// Mitsubishi GX Works2 project: BluestarPlc 17-06-2023f1   PLC: Q03UDV

PROGRAM MAIN
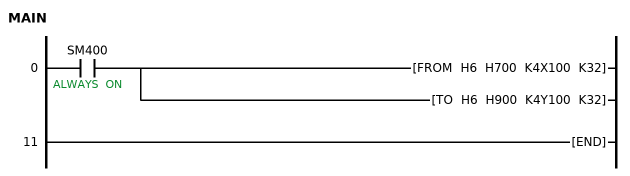
0     LD      SM400  ; ALWAYS  ON
      FROM    H6 H700 K4X100 K32  ; DO1_CMD_ENBLE
      TO      H6 H900 K4Y100 K32  ; DI01_IMSTP
11    END
END_PROGRAM

PROGRAM LOGIC
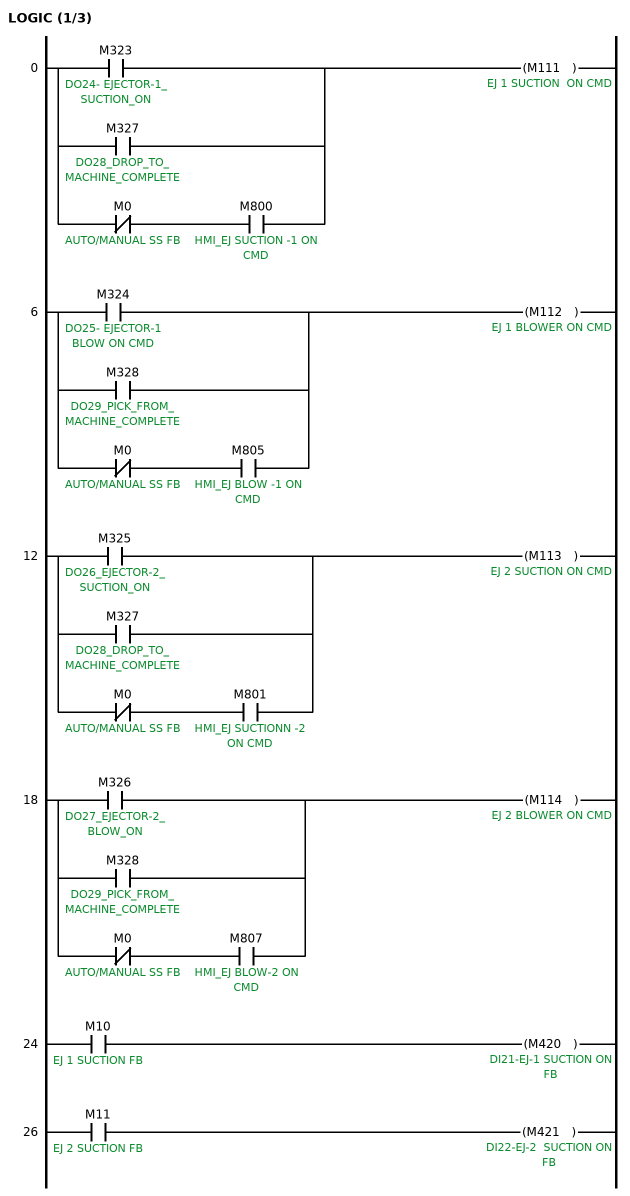
0     LD      M323  ; DO24- EJECTOR-1_SUCTION_ON
      OR      M327  ; DO28_DROP_TO_MACHINE_COMPLETE
      LDI     M0  ; AUTO/MANUAL SS FB
      AND     M800  ; HMI_EJ SUCTION -1 ON CMD
      ORB
      OUT     M111  ; EJ 1 SUCTION  ON CMD
6     LD      M324  ; DO25- EJECTOR-1  BLOW ON CMD
      OR      M328  ; DO29_PICK_FROM_MACHINE_COMPLETE
      LDI     M0  ; AUTO/MANUAL SS FB
      AND     M805  ; HMI_EJ BLOW -1 ON CMD
      ORB
      OUT     M112  ; EJ 1 BLOWER ON CMD
12    LD      M325  ; DO26_EJECTOR-2_SUCTION_ON
      OR      M327  ; DO28_DROP_TO_MACHINE_COMPLETE
      LDI     M0  ; AUTO/MANUAL SS FB
      AND     M801  ; HMI_EJ SUCTIONN -2 ON CMD
      ORB
      OUT     M113  ; EJ 2 SUCTION ON CMD
18    LD      M326  ; DO27_EJECTOR-2_BLOW_ON
      OR      M328  ; DO29_PICK_FROM_MACHINE_COMPLETE
      LDI     M0  ; AUTO/MANUAL SS FB
      AND     M807  ; HMI_EJ BLOW-2 ON CMD
      ORB
      OUT     M114  ; EJ 2 BLOWER ON CMD
24    LD      M10  ; EJ 1 SUCTION FB
      OUT     M420  ; DI21-EJ-1 SUCTION ON FB
26    LD      M11  ; EJ 2 SUCTION FB
      OUT     M421  ; DI22-EJ-2  SUCTION ON FB
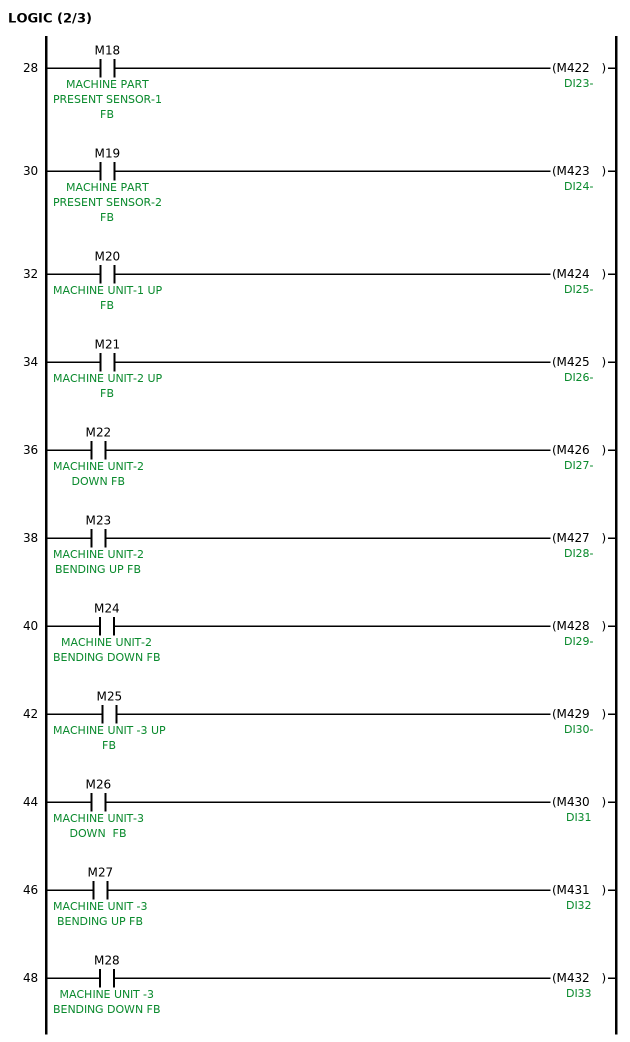
28    LD      M18  ; MACHINE PART PRESENT SENSOR-1 FB
      OUT     M422  ; DI23-
30    LD      M19  ; MACHINE PART PRESENT SENSOR-2 FB
      OUT     M423  ; DI24-
32    LD      M20  ; MACHINE UNIT-1 UP FB
      OUT     M424  ; DI25-
34    LD      M21  ; MACHINE UNIT-2 UP FB
      OUT     M425  ; DI26-
36    LD      M22  ; MACHINE UNIT-2 DOWN FB
      OUT     M426  ; DI27-
38    LD      M23  ; MACHINE UNIT-2 BENDING UP FB
      OUT     M427  ; DI28-
40    LD      M24  ; MACHINE UNIT-2 BENDING DOWN FB
      OUT     M428  ; DI29-
42    LD      M25  ; MACHINE UNIT -3 UP FB
      OUT     M429  ; DI30-
44    LD      M26  ; MACHINE UNIT-3 DOWN  FB
      OUT     M430  ; DI31
46    LD      M27  ; MACHINE UNIT -3 BENDING UP FB
      OUT     M431  ; DI32
48    LD      M28  ; MACHINE UNIT -3 BENDING DOWN FB
      OUT     M432  ; DI33
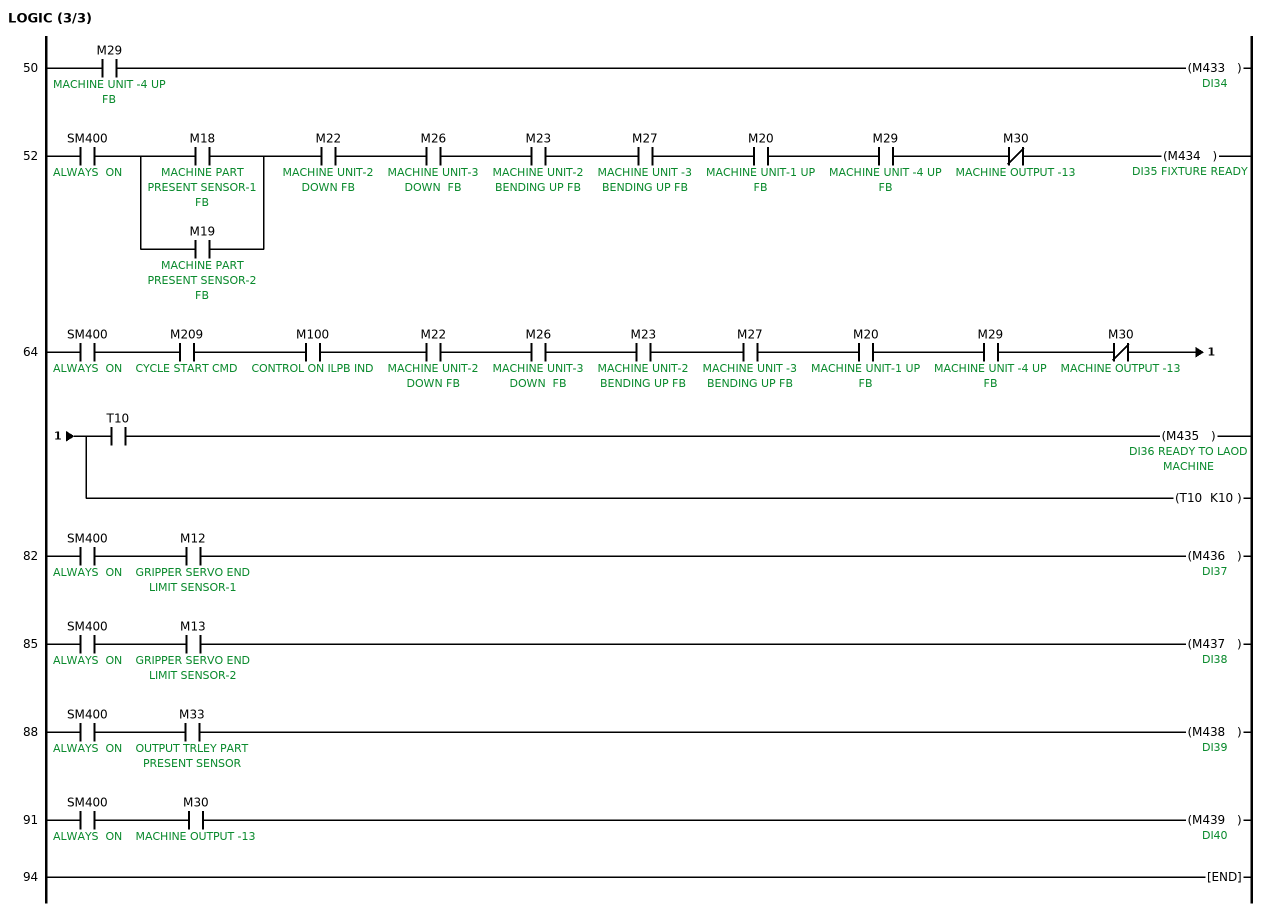
50    LD      M29  ; MACHINE UNIT -4 UP FB
      OUT     M433  ; DI34
52    LD      SM400  ; ALWAYS  ON
      LD      M18  ; MACHINE PART PRESENT SENSOR-1 FB
      OR      M19  ; MACHINE PART PRESENT SENSOR-2 FB
      ANB
      AND     M22  ; MACHINE UNIT-2 DOWN FB
      AND     M26  ; MACHINE UNIT-3 DOWN  FB
      AND     M23  ; MACHINE UNIT-2 BENDING UP FB
      AND     M27  ; MACHINE UNIT -3 BENDING UP FB
      AND     M20  ; MACHINE UNIT-1 UP FB
      AND     M29  ; MACHINE UNIT -4 UP FB
      ANI     M30  ; MACHINE OUTPUT -13
      OUT     M434  ; DI35 FIXTURE READY
64    LD      SM400  ; ALWAYS  ON
      AND     M209  ; CYCLE START CMD
      AND     M100  ; CONTROL ON ILPB IND
      AND     M22  ; MACHINE UNIT-2 DOWN FB
      AND     M26  ; MACHINE UNIT-3 DOWN  FB
      AND     M23  ; MACHINE UNIT-2 BENDING UP FB
      AND     M27  ; MACHINE UNIT -3 BENDING UP FB
      AND     M20  ; MACHINE UNIT-1 UP FB
      AND     M29  ; MACHINE UNIT -4 UP FB
      ANI     M30  ; MACHINE OUTPUT -13
      MPS
      AND     T10
      OUT     M435  ; DI36 READY TO LAOD MACHINE
      MPP
      OUT     T10 K10
82    LD      SM400  ; ALWAYS  ON
      AND     M12  ; GRIPPER SERVO END LIMIT SENSOR-1
      OUT     M436  ; DI37
85    LD      SM400  ; ALWAYS  ON
      AND     M13  ; GRIPPER SERVO END LIMIT SENSOR-2
      OUT     M437  ; DI38
88    LD      SM400  ; ALWAYS  ON
      AND     M33  ; OUTPUT TRLEY PART PRESENT SENSOR
      OUT     M438  ; DI39
91    LD      SM400  ; ALWAYS  ON
      AND     M30  ; MACHINE OUTPUT -13
      OUT     M439  ; DI40
94    END
END_PROGRAM

PROGRAM D-NET
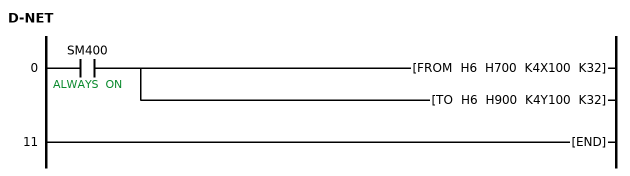
0     LD      SM400  ; ALWAYS  ON
      FROM    H6 H700 K4X100 K32  ; DO1_CMD_ENBLE
      TO      H6 H900 K4Y100 K32  ; DI01_IMSTP
11    END
END_PROGRAM

PROGRAM RBT-IN
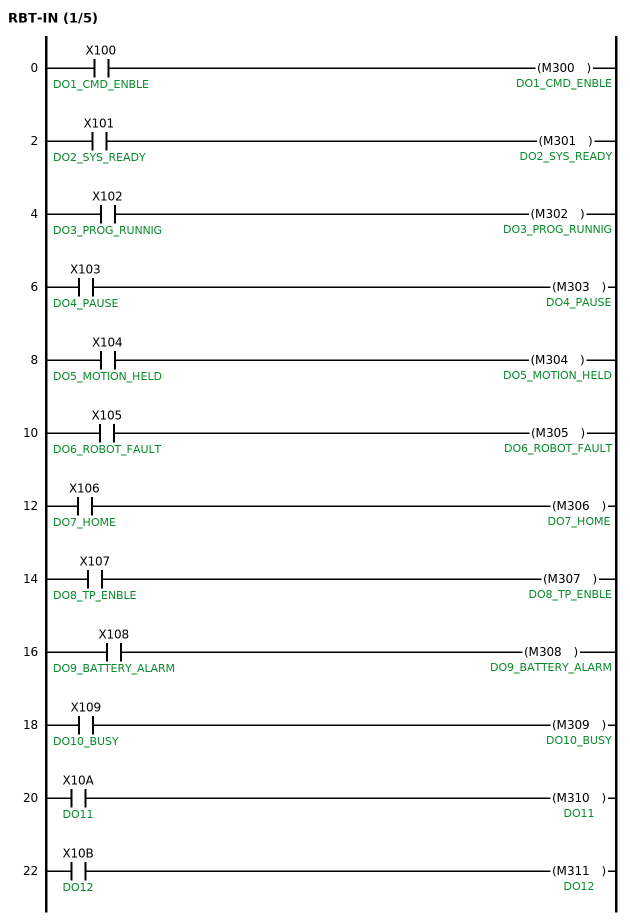
0     LD      X100  ; DO1_CMD_ENBLE
      OUT     M300  ; DO1_CMD_ENBLE
2     LD      X101  ; DO2_SYS_READY
      OUT     M301  ; DO2_SYS_READY
4     LD      X102  ; DO3_PROG_RUNNIG
      OUT     M302  ; DO3_PROG_RUNNIG
6     LD      X103  ; DO4_PAUSE
      OUT     M303  ; DO4_PAUSE
8     LD      X104  ; DO5_MOTION_HELD
      OUT     M304  ; DO5_MOTION_HELD
10    LD      X105  ; DO6_ROBOT_FAULT
      OUT     M305  ; DO6_ROBOT_FAULT
12    LD      X106  ; DO7_HOME
      OUT     M306  ; DO7_HOME
14    LD      X107  ; DO8_TP_ENBLE
      OUT     M307  ; DO8_TP_ENBLE
16    LD      X108  ; DO9_BATTERY_ALARM
      OUT     M308  ; DO9_BATTERY_ALARM
18    LD      X109  ; DO10_BUSY
      OUT     M309  ; DO10_BUSY
20    LD      X10A  ; DO11
      OUT     M310  ; DO11
22    LD      X10B  ; DO12
      OUT     M311  ; DO12
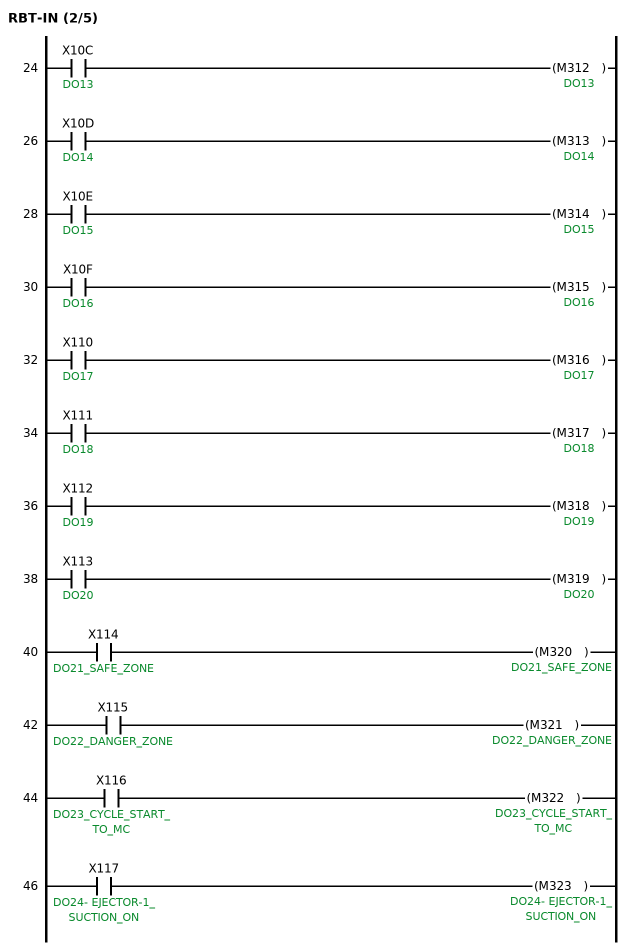
24    LD      X10C  ; DO13
      OUT     M312  ; DO13
26    LD      X10D  ; DO14
      OUT     M313  ; DO14
28    LD      X10E  ; DO15
      OUT     M314  ; DO15
30    LD      X10F  ; DO16
      OUT     M315  ; DO16
32    LD      X110  ; DO17
      OUT     M316  ; DO17
34    LD      X111  ; DO18
      OUT     M317  ; DO18
36    LD      X112  ; DO19
      OUT     M318  ; DO19
38    LD      X113  ; DO20
      OUT     M319  ; DO20
40    LD      X114  ; DO21_SAFE_ZONE
      OUT     M320  ; DO21_SAFE_ZONE
42    LD      X115  ; DO22_DANGER_ZONE
      OUT     M321  ; DO22_DANGER_ZONE
44    LD      X116  ; DO23_CYCLE_START_TO_MC
      OUT     M322  ; DO23_CYCLE_START_TO_MC
46    LD      X117  ; DO24- EJECTOR-1_SUCTION_ON
      OUT     M323  ; DO24- EJECTOR-1_SUCTION_ON
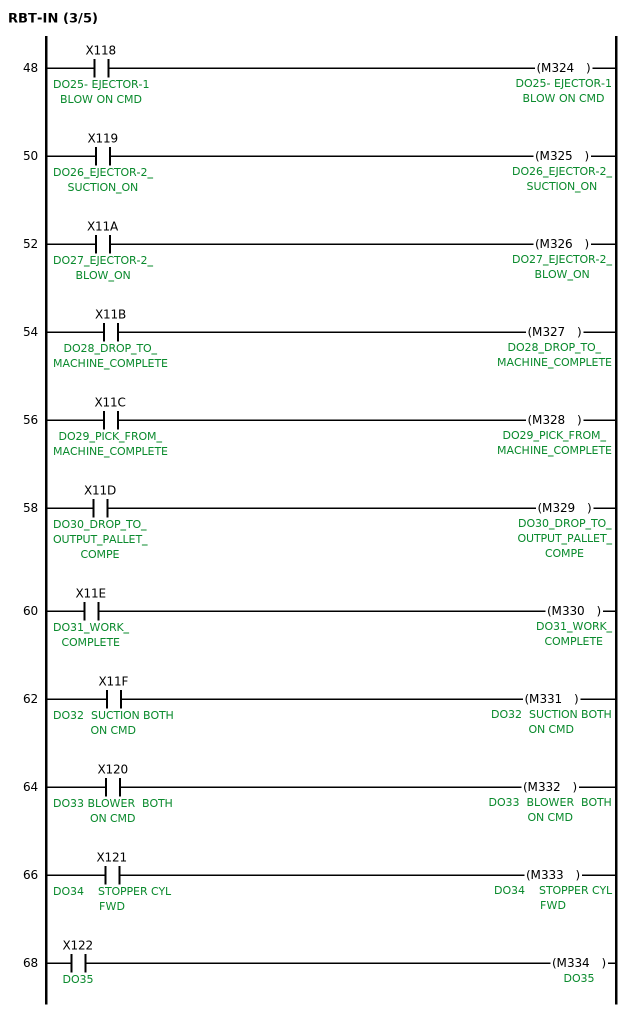
48    LD      X118  ; DO25- EJECTOR-1  BLOW ON CMD
      OUT     M324  ; DO25- EJECTOR-1  BLOW ON CMD
50    LD      X119  ; DO26_EJECTOR-2_SUCTION_ON
      OUT     M325  ; DO26_EJECTOR-2_SUCTION_ON
52    LD      X11A  ; DO27_EJECTOR-2_BLOW_ON
      OUT     M326  ; DO27_EJECTOR-2_BLOW_ON
54    LD      X11B  ; DO28_DROP_TO_MACHINE_COMPLETE
      OUT     M327  ; DO28_DROP_TO_MACHINE_COMPLETE
56    LD      X11C  ; DO29_PICK_FROM_MACHINE_COMPLETE
      OUT     M328  ; DO29_PICK_FROM_MACHINE_COMPLETE
58    LD      X11D  ; DO30_DROP_TO_OUTPUT_PALLET_COMPE
      OUT     M329  ; DO30_DROP_TO_OUTPUT_PALLET_COMPE
60    LD      X11E  ; DO31_WORK_COMPLETE
      OUT     M330  ; DO31_WORK_COMPLETE
62    LD      X11F  ; DO32  SUCTION BOTH ON CMD
      OUT     M331  ; DO32  SUCTION BOTH ON CMD
64    LD      X120  ; DO33 BLOWER  BOTH ON CMD
      OUT     M332  ; DO33  BLOWER  BOTH ON CMD
66    LD      X121  ; DO34    STOPPER CYL FWD
      OUT     M333  ; DO34    STOPPER CYL FWD
68    LD      X122  ; DO35
      OUT     M334  ; DO35
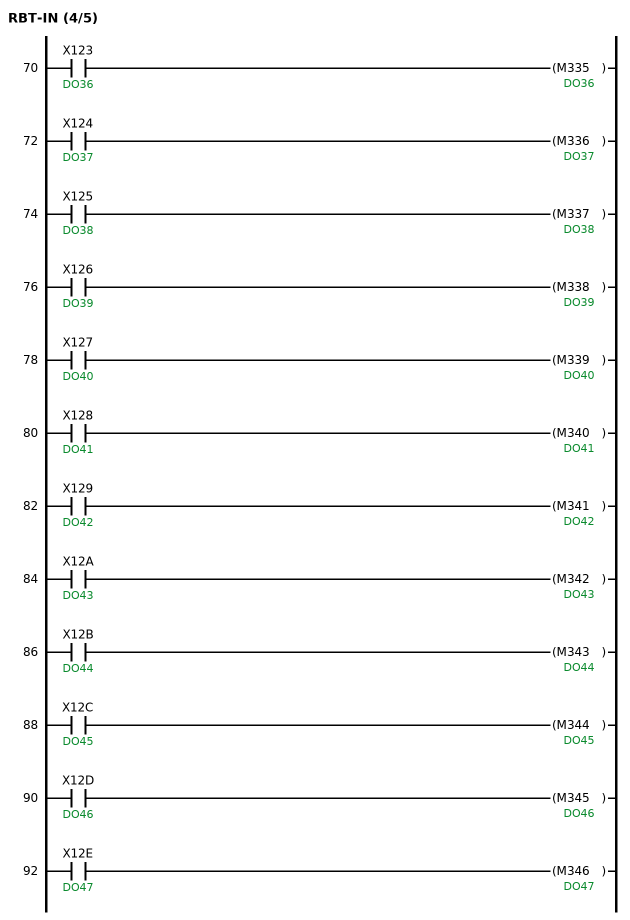
70    LD      X123  ; DO36
      OUT     M335  ; DO36
72    LD      X124  ; DO37
      OUT     M336  ; DO37
74    LD      X125  ; DO38
      OUT     M337  ; DO38
76    LD      X126  ; DO39
      OUT     M338  ; DO39
78    LD      X127  ; DO40
      OUT     M339  ; DO40
80    LD      X128  ; DO41
      OUT     M340  ; DO41
82    LD      X129  ; DO42
      OUT     M341  ; DO42
84    LD      X12A  ; DO43
      OUT     M342  ; DO43
86    LD      X12B  ; DO44
      OUT     M343  ; DO44
88    LD      X12C  ; DO45
      OUT     M344  ; DO45
90    LD      X12D  ; DO46
      OUT     M345  ; DO46
92    LD      X12E  ; DO47
      OUT     M346  ; DO47
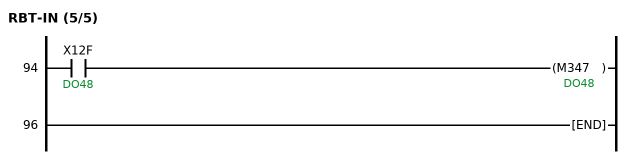
94    LD      X12F  ; DO48
      OUT     M347  ; DO48
96    END
END_PROGRAM

PROGRAM RBT-OUT
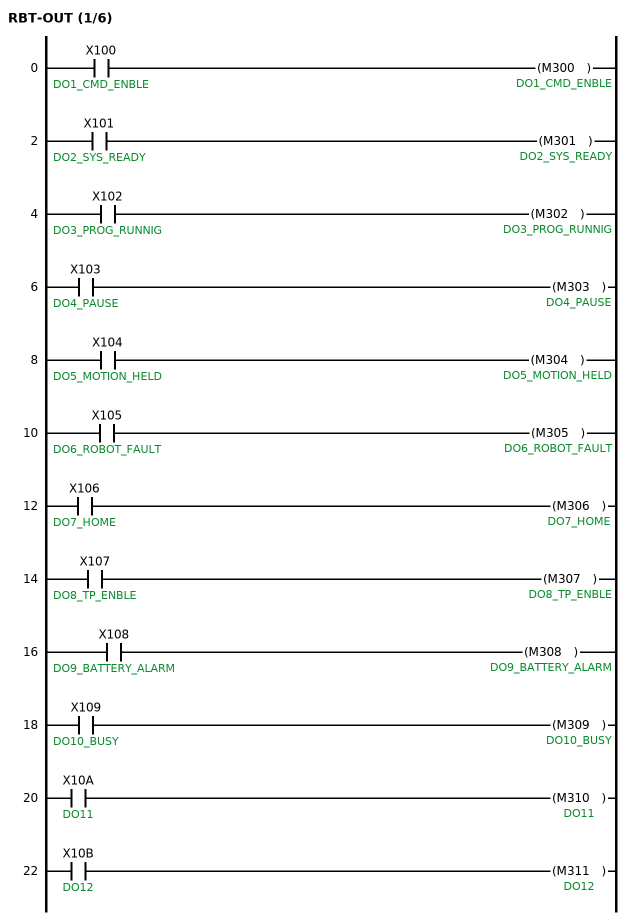
0     LD      X100  ; DO1_CMD_ENBLE
      OUT     M300  ; DO1_CMD_ENBLE
2     LD      X101  ; DO2_SYS_READY
      OUT     M301  ; DO2_SYS_READY
4     LD      X102  ; DO3_PROG_RUNNIG
      OUT     M302  ; DO3_PROG_RUNNIG
6     LD      X103  ; DO4_PAUSE
      OUT     M303  ; DO4_PAUSE
8     LD      X104  ; DO5_MOTION_HELD
      OUT     M304  ; DO5_MOTION_HELD
10    LD      X105  ; DO6_ROBOT_FAULT
      OUT     M305  ; DO6_ROBOT_FAULT
12    LD      X106  ; DO7_HOME
      OUT     M306  ; DO7_HOME
14    LD      X107  ; DO8_TP_ENBLE
      OUT     M307  ; DO8_TP_ENBLE
16    LD      X108  ; DO9_BATTERY_ALARM
      OUT     M308  ; DO9_BATTERY_ALARM
18    LD      X109  ; DO10_BUSY
      OUT     M309  ; DO10_BUSY
20    LD      X10A  ; DO11
      OUT     M310  ; DO11
22    LD      X10B  ; DO12
      OUT     M311  ; DO12
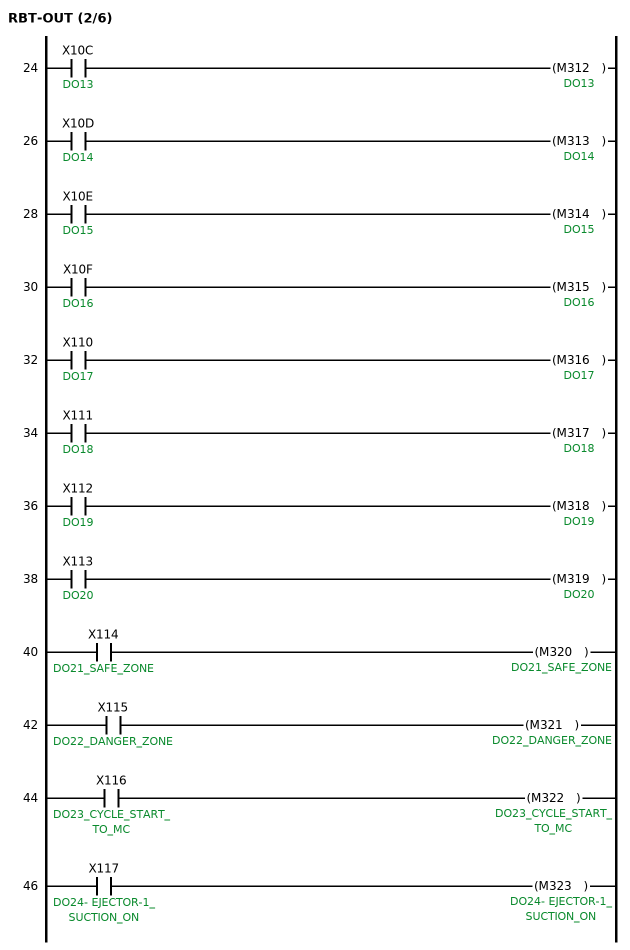
24    LD      X10C  ; DO13
      OUT     M312  ; DO13
26    LD      X10D  ; DO14
      OUT     M313  ; DO14
28    LD      X10E  ; DO15
      OUT     M314  ; DO15
30    LD      X10F  ; DO16
      OUT     M315  ; DO16
32    LD      X110  ; DO17
      OUT     M316  ; DO17
34    LD      X111  ; DO18
      OUT     M317  ; DO18
36    LD      X112  ; DO19
      OUT     M318  ; DO19
38    LD      X113  ; DO20
      OUT     M319  ; DO20
40    LD      X114  ; DO21_SAFE_ZONE
      OUT     M320  ; DO21_SAFE_ZONE
42    LD      X115  ; DO22_DANGER_ZONE
      OUT     M321  ; DO22_DANGER_ZONE
44    LD      X116  ; DO23_CYCLE_START_TO_MC
      OUT     M322  ; DO23_CYCLE_START_TO_MC
46    LD      X117  ; DO24- EJECTOR-1_SUCTION_ON
      OUT     M323  ; DO24- EJECTOR-1_SUCTION_ON
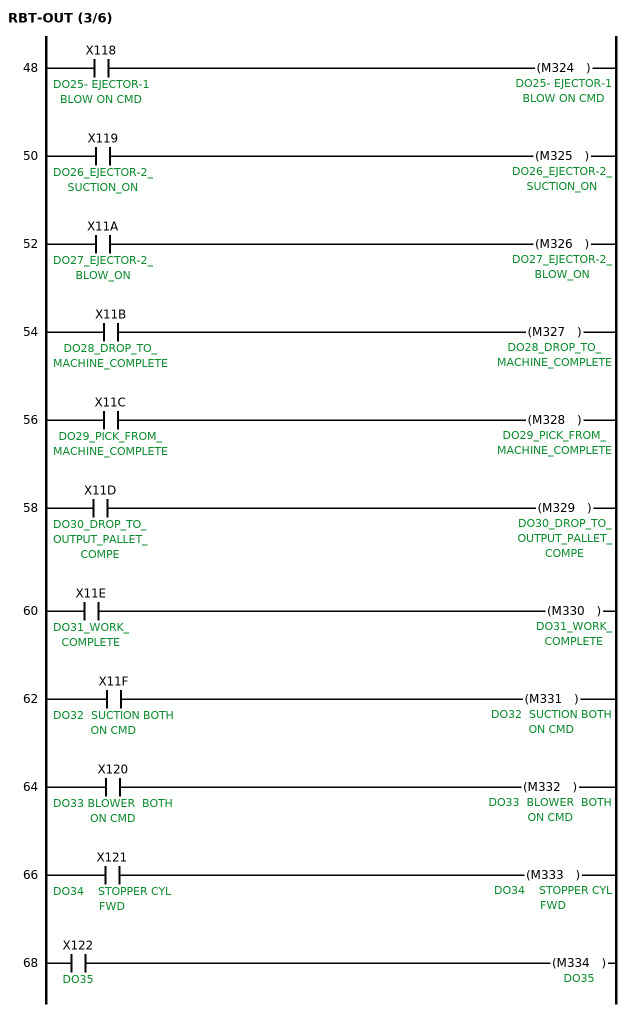
48    LD      X118  ; DO25- EJECTOR-1  BLOW ON CMD
      OUT     M324  ; DO25- EJECTOR-1  BLOW ON CMD
50    LD      X119  ; DO26_EJECTOR-2_SUCTION_ON
      OUT     M325  ; DO26_EJECTOR-2_SUCTION_ON
52    LD      X11A  ; DO27_EJECTOR-2_BLOW_ON
      OUT     M326  ; DO27_EJECTOR-2_BLOW_ON
54    LD      X11B  ; DO28_DROP_TO_MACHINE_COMPLETE
      OUT     M327  ; DO28_DROP_TO_MACHINE_COMPLETE
56    LD      X11C  ; DO29_PICK_FROM_MACHINE_COMPLETE
      OUT     M328  ; DO29_PICK_FROM_MACHINE_COMPLETE
58    LD      X11D  ; DO30_DROP_TO_OUTPUT_PALLET_COMPE
      OUT     M329  ; DO30_DROP_TO_OUTPUT_PALLET_COMPE
60    LD      X11E  ; DO31_WORK_COMPLETE
      OUT     M330  ; DO31_WORK_COMPLETE
62    LD      X11F  ; DO32  SUCTION BOTH ON CMD
      OUT     M331  ; DO32  SUCTION BOTH ON CMD
64    LD      X120  ; DO33 BLOWER  BOTH ON CMD
      OUT     M332  ; DO33  BLOWER  BOTH ON CMD
66    LD      X121  ; DO34    STOPPER CYL FWD
      OUT     M333  ; DO34    STOPPER CYL FWD
68    LD      X122  ; DO35
      OUT     M334  ; DO35
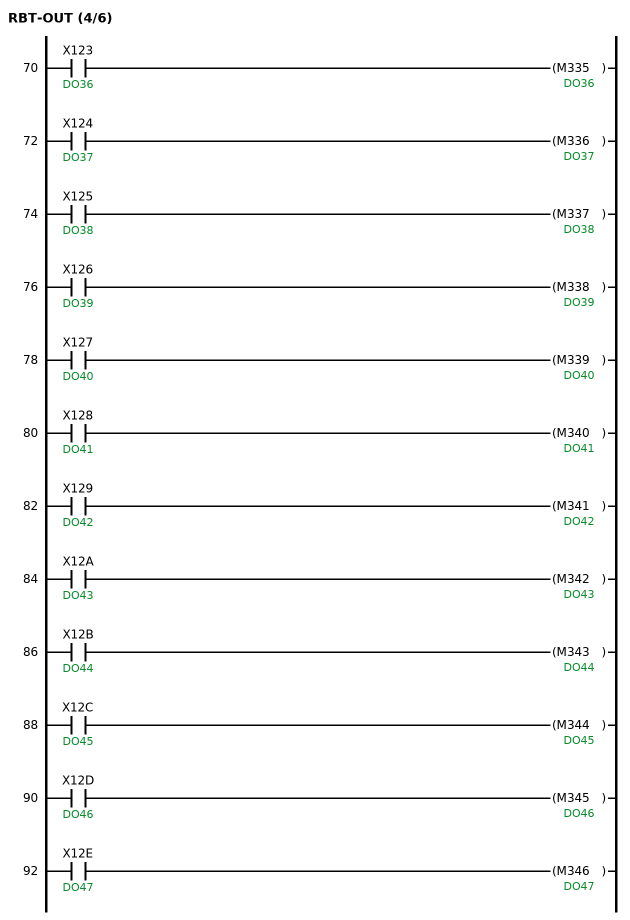
70    LD      X123  ; DO36
      OUT     M335  ; DO36
72    LD      X124  ; DO37
      OUT     M336  ; DO37
74    LD      X125  ; DO38
      OUT     M337  ; DO38
76    LD      X126  ; DO39
      OUT     M338  ; DO39
78    LD      X127  ; DO40
      OUT     M339  ; DO40
80    LD      X128  ; DO41
      OUT     M340  ; DO41
82    LD      X129  ; DO42
      OUT     M341  ; DO42
84    LD      X12A  ; DO43
      OUT     M342  ; DO43
86    LD      X12B  ; DO44
      OUT     M343  ; DO44
88    LD      X12C  ; DO45
      OUT     M344  ; DO45
90    LD      X12D  ; DO46
      OUT     M345  ; DO46
92    LD      X12E  ; DO47
      OUT     M346  ; DO47
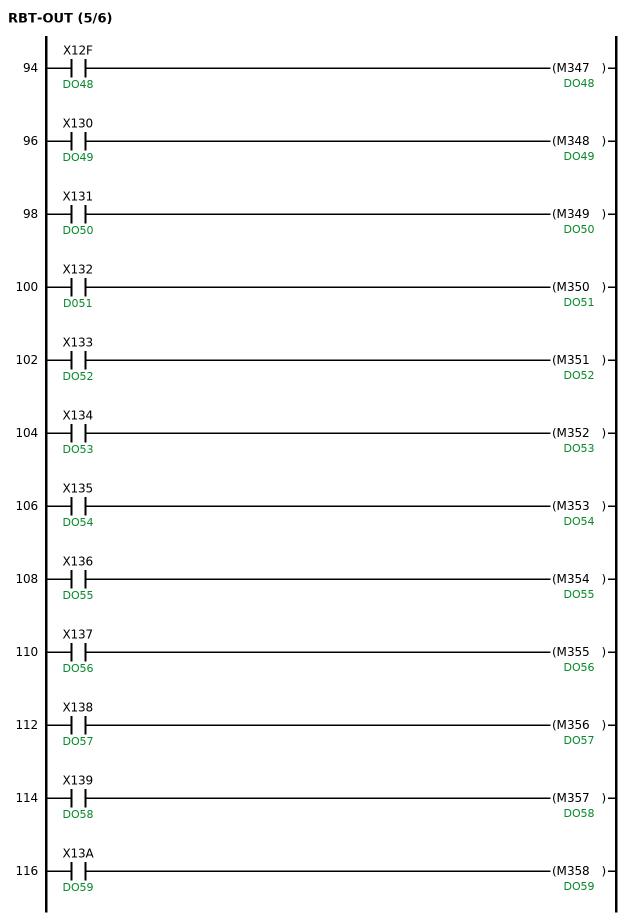
94    LD      X12F  ; DO48
      OUT     M347  ; DO48
96    LD      X130  ; DO49
      OUT     M348  ; DO49
98    LD      X131  ; DO50
      OUT     M349  ; DO50
100   LD      X132  ; D051
      OUT     M350  ; DO51
102   LD      X133  ; DO52
      OUT     M351  ; DO52
104   LD      X134  ; DO53
      OUT     M352  ; DO53
106   LD      X135  ; DO54
      OUT     M353  ; DO54
108   LD      X136  ; DO55
      OUT     M354  ; DO55
110   LD      X137  ; DO56
      OUT     M355  ; DO56
112   LD      X138  ; DO57
      OUT     M356  ; DO57
114   LD      X139  ; DO58
      OUT     M357  ; DO58
116   LD      X13A  ; DO59
      OUT     M358  ; DO59
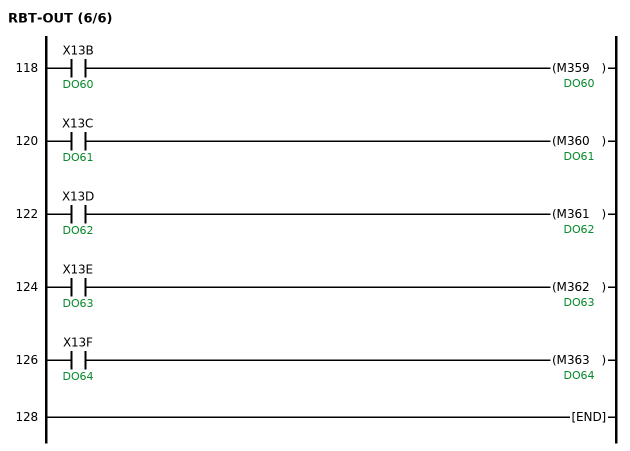
118   LD      X13B  ; DO60
      OUT     M359  ; DO60
120   LD      X13C  ; DO61
      OUT     M360  ; DO61
122   LD      X13D  ; DO62
      OUT     M361  ; DO62
124   LD      X13E  ; DO63
      OUT     M362  ; DO63
126   LD      X13F  ; DO64
      OUT     M363  ; DO64
128   END
END_PROGRAM

PROGRAM PLC-IN
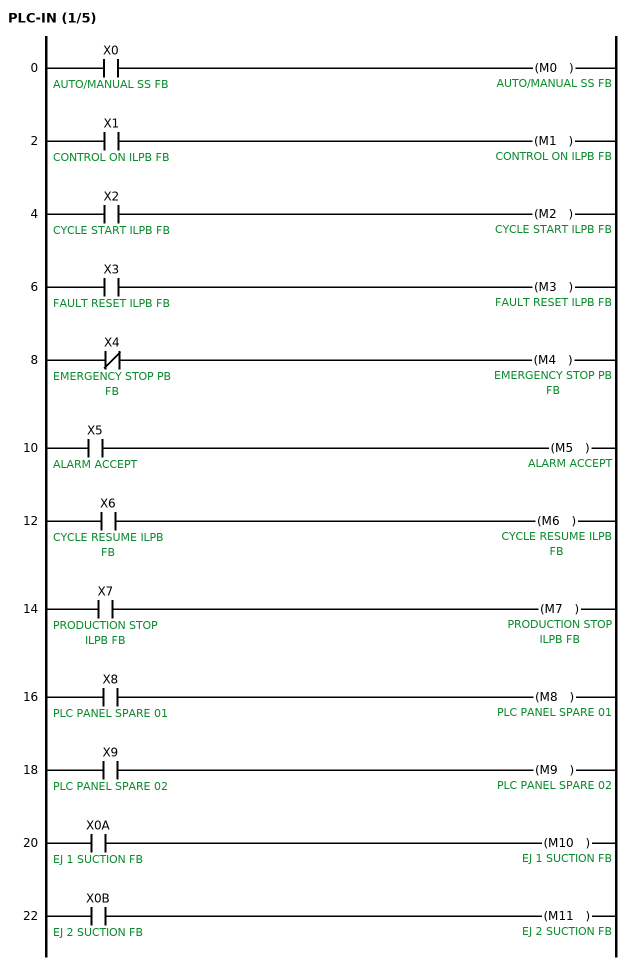
0     LD      X0  ; AUTO/MANUAL SS FB
      OUT     M0  ; AUTO/MANUAL SS FB
2     LD      X1  ; CONTROL ON ILPB FB
      OUT     M1  ; CONTROL ON ILPB FB
4     LD      X2  ; CYCLE START ILPB FB
      OUT     M2  ; CYCLE START ILPB FB
6     LD      X3  ; FAULT RESET ILPB FB
      OUT     M3  ; FAULT RESET ILPB FB
8     LDI     X4  ; EMERGENCY STOP PB FB
      OUT     M4  ; EMERGENCY STOP PB FB
10    LD      X5  ; ALARM ACCEPT
      OUT     M5  ; ALARM ACCEPT
12    LD      X6  ; CYCLE RESUME ILPB FB
      OUT     M6  ; CYCLE RESUME ILPB FB
14    LD      X7  ; PRODUCTION STOP ILPB FB
      OUT     M7  ; PRODUCTION STOP ILPB FB
16    LD      X8  ; PLC PANEL SPARE 01
      OUT     M8  ; PLC PANEL SPARE 01
18    LD      X9  ; PLC PANEL SPARE 02
      OUT     M9  ; PLC PANEL SPARE 02
20    LD      X0A  ; EJ 1 SUCTION FB
      OUT     M10  ; EJ 1 SUCTION FB
22    LD      X0B  ; EJ 2 SUCTION FB
      OUT     M11  ; EJ 2 SUCTION FB
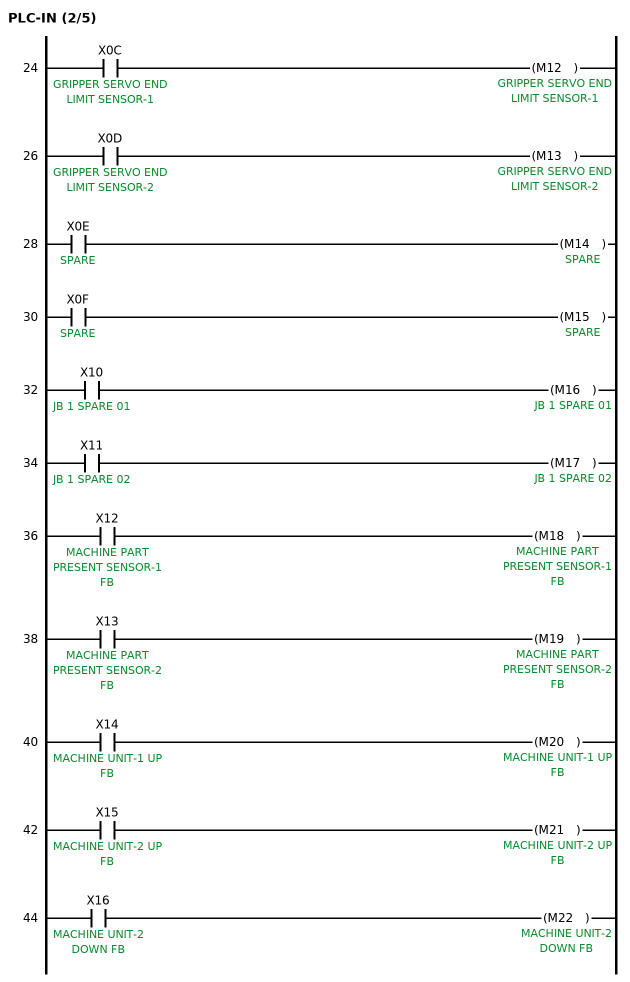
24    LD      X0C  ; GRIPPER SERVO END LIMIT SENSOR-1
      OUT     M12  ; GRIPPER SERVO END LIMIT SENSOR-1
26    LD      X0D  ; GRIPPER SERVO END LIMIT SENSOR-2
      OUT     M13  ; GRIPPER SERVO END LIMIT SENSOR-2
28    LD      X0E  ; SPARE
      OUT     M14  ; SPARE
30    LD      X0F  ; SPARE
      OUT     M15  ; SPARE
32    LD      X10  ; JB 1 SPARE 01
      OUT     M16  ; JB 1 SPARE 01
34    LD      X11  ; JB 1 SPARE 02
      OUT     M17  ; JB 1 SPARE 02
36    LD      X12  ; MACHINE PART PRESENT SENSOR-1 FB
      OUT     M18  ; MACHINE PART PRESENT SENSOR-1 FB
38    LD      X13  ; MACHINE PART PRESENT SENSOR-2 FB
      OUT     M19  ; MACHINE PART PRESENT SENSOR-2 FB
40    LD      X14  ; MACHINE UNIT-1 UP FB
      OUT     M20  ; MACHINE UNIT-1 UP FB
42    LD      X15  ; MACHINE UNIT-2 UP FB
      OUT     M21  ; MACHINE UNIT-2 UP FB
44    LD      X16  ; MACHINE UNIT-2 DOWN FB
      OUT     M22  ; MACHINE UNIT-2 DOWN FB
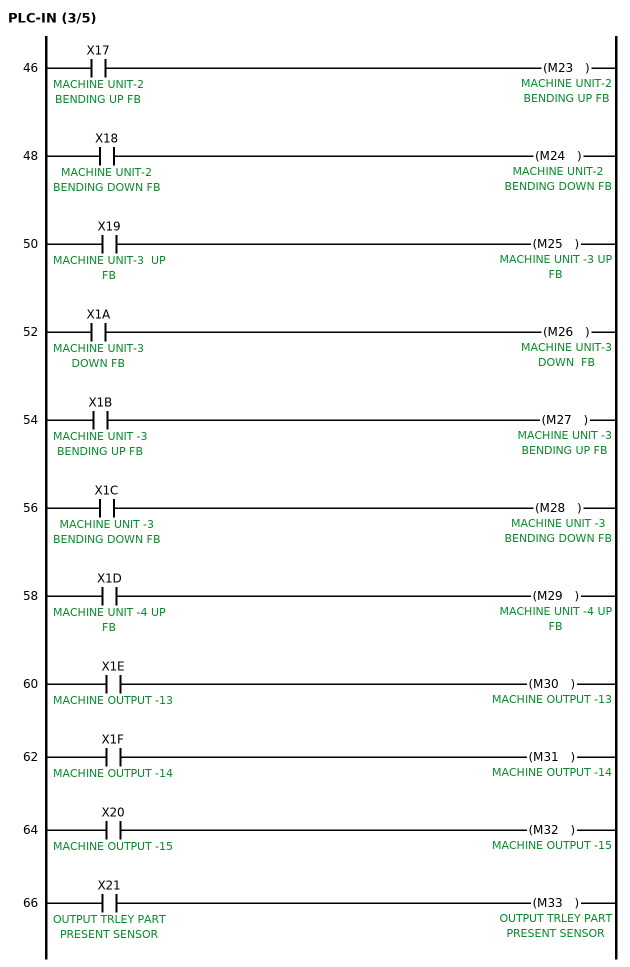
46    LD      X17  ; MACHINE UNIT-2 BENDING UP FB
      OUT     M23  ; MACHINE UNIT-2 BENDING UP FB
48    LD      X18  ; MACHINE UNIT-2 BENDING DOWN FB
      OUT     M24  ; MACHINE UNIT-2 BENDING DOWN FB
50    LD      X19  ; MACHINE UNIT-3  UP FB
      OUT     M25  ; MACHINE UNIT -3 UP FB
52    LD      X1A  ; MACHINE UNIT-3 DOWN FB
      OUT     M26  ; MACHINE UNIT-3 DOWN  FB
54    LD      X1B  ; MACHINE UNIT -3 BENDING UP FB
      OUT     M27  ; MACHINE UNIT -3 BENDING UP FB
56    LD      X1C  ; MACHINE UNIT -3 BENDING DOWN FB
      OUT     M28  ; MACHINE UNIT -3 BENDING DOWN FB
58    LD      X1D  ; MACHINE UNIT -4 UP FB
      OUT     M29  ; MACHINE UNIT -4 UP FB
60    LD      X1E  ; MACHINE OUTPUT -13
      OUT     M30  ; MACHINE OUTPUT -13
62    LD      X1F  ; MACHINE OUTPUT -14
      OUT     M31  ; MACHINE OUTPUT -14
64    LD      X20  ; MACHINE OUTPUT -15
      OUT     M32  ; MACHINE OUTPUT -15
66    LD      X21  ; OUTPUT TRLEY PART PRESENT SENSOR
      OUT     M33  ; OUTPUT TRLEY PART PRESENT SENSOR
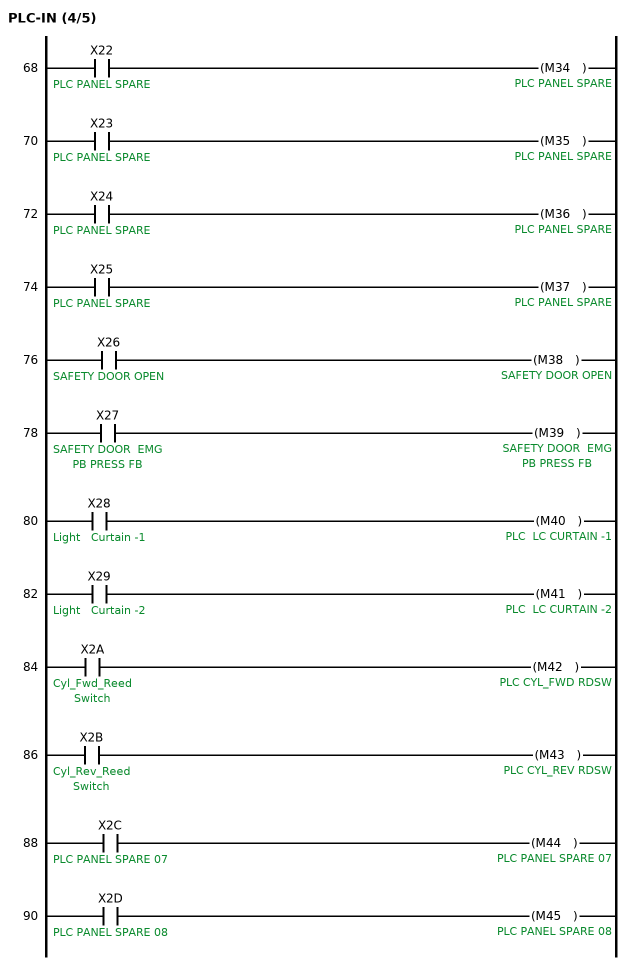
68    LD      X22  ; PLC PANEL SPARE
      OUT     M34  ; PLC PANEL SPARE
70    LD      X23  ; PLC PANEL SPARE
      OUT     M35  ; PLC PANEL SPARE
72    LD      X24  ; PLC PANEL SPARE
      OUT     M36  ; PLC PANEL SPARE
74    LD      X25  ; PLC PANEL SPARE
      OUT     M37  ; PLC PANEL SPARE
76    LD      X26  ; SAFETY DOOR OPEN
      OUT     M38  ; SAFETY DOOR OPEN
78    LD      X27  ; SAFETY DOOR  EMG PB PRESS FB
      OUT     M39  ; SAFETY DOOR  EMG PB PRESS FB
80    LD      X28  ; Light   Curtain -1
      OUT     M40  ; PLC  LC CURTAIN -1
82    LD      X29  ; Light   Curtain -2
      OUT     M41  ; PLC  LC CURTAIN -2
84    LD      X2A  ; Cyl_Fwd_Reed    Switch
      OUT     M42  ; PLC CYL_FWD RDSW
86    LD      X2B  ; Cyl_Rev_Reed    Switch
      OUT     M43  ; PLC CYL_REV RDSW
88    LD      X2C  ; PLC PANEL SPARE 07
      OUT     M44  ; PLC PANEL SPARE 07
90    LD      X2D  ; PLC PANEL SPARE 08
      OUT     M45  ; PLC PANEL SPARE 08
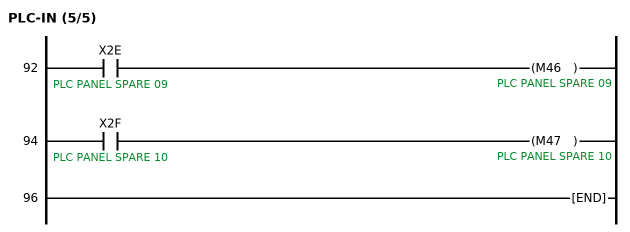
92    LD      X2E  ; PLC PANEL SPARE 09
      OUT     M46  ; PLC PANEL SPARE 09
94    LD      X2F  ; PLC PANEL SPARE 10
      OUT     M47  ; PLC PANEL SPARE 10
96    END
END_PROGRAM

PROGRAM PLC-OUT
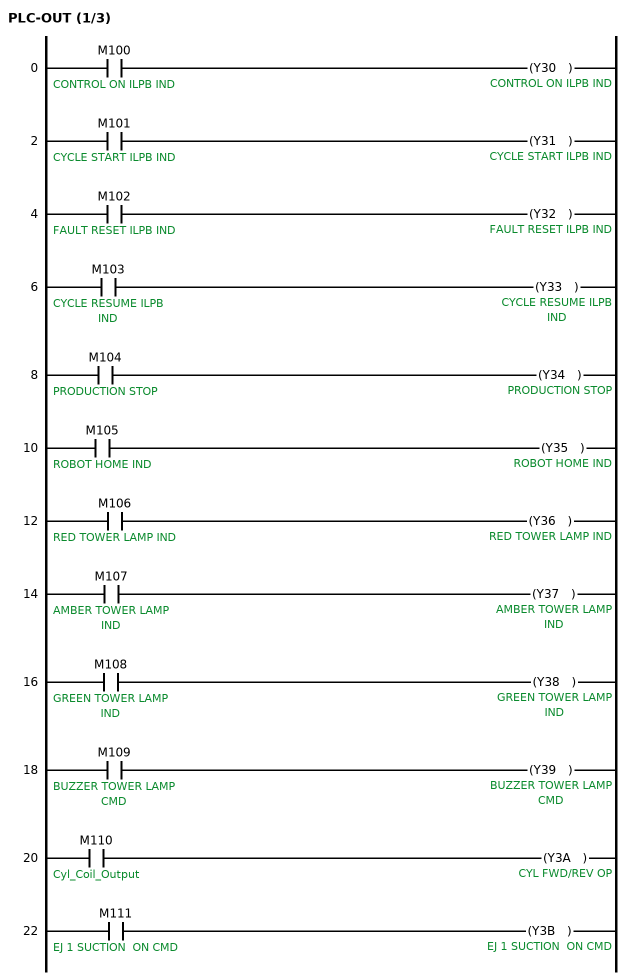
0     LD      M100  ; CONTROL ON ILPB IND
      OUT     Y30  ; CONTROL ON ILPB IND
2     LD      M101  ; CYCLE START ILPB IND
      OUT     Y31  ; CYCLE START ILPB IND
4     LD      M102  ; FAULT RESET ILPB IND
      OUT     Y32  ; FAULT RESET ILPB IND
6     LD      M103  ; CYCLE RESUME ILPB IND
      OUT     Y33  ; CYCLE RESUME ILPB IND
8     LD      M104  ; PRODUCTION STOP
      OUT     Y34  ; PRODUCTION STOP
10    LD      M105  ; ROBOT HOME IND
      OUT     Y35  ; ROBOT HOME IND
12    LD      M106  ; RED TOWER LAMP IND
      OUT     Y36  ; RED TOWER LAMP IND
14    LD      M107  ; AMBER TOWER LAMP IND
      OUT     Y37  ; AMBER TOWER LAMP IND
16    LD      M108  ; GREEN TOWER LAMP IND
      OUT     Y38  ; GREEN TOWER LAMP IND
18    LD      M109  ; BUZZER TOWER LAMP CMD
      OUT     Y39  ; BUZZER TOWER LAMP CMD
20    LD      M110  ; Cyl_Coil_Output
      OUT     Y3A  ; CYL FWD/REV OP
22    LD      M111  ; EJ 1 SUCTION  ON CMD
      OUT     Y3B  ; EJ 1 SUCTION  ON CMD
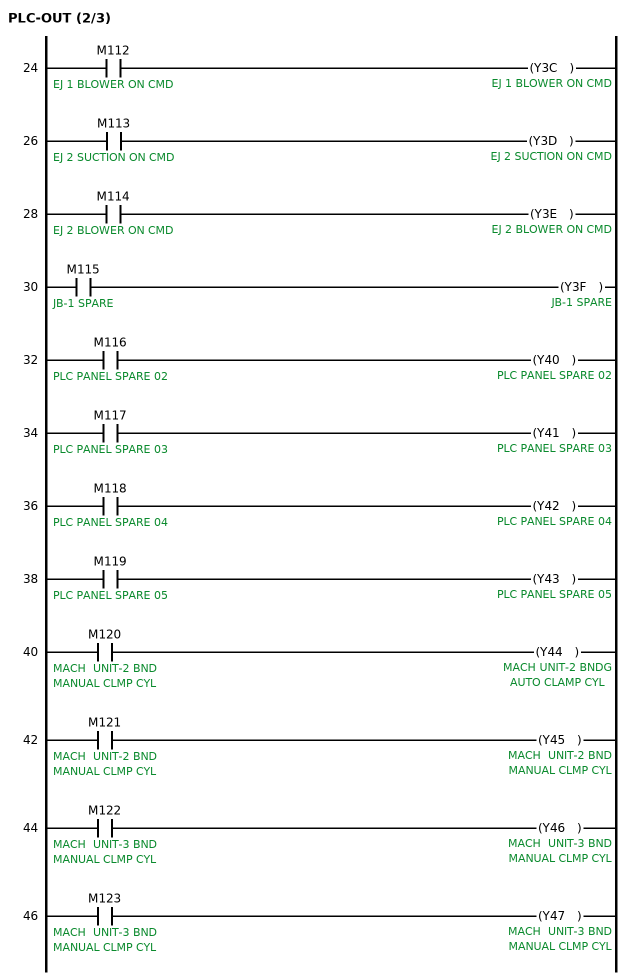
24    LD      M112  ; EJ 1 BLOWER ON CMD
      OUT     Y3C  ; EJ 1 BLOWER ON CMD
26    LD      M113  ; EJ 2 SUCTION ON CMD
      OUT     Y3D  ; EJ 2 SUCTION ON CMD
28    LD      M114  ; EJ 2 BLOWER ON CMD
      OUT     Y3E  ; EJ 2 BLOWER ON CMD
30    LD      M115  ; JB-1 SPARE
      OUT     Y3F  ; JB-1 SPARE
32    LD      M116  ; PLC PANEL SPARE 02
      OUT     Y40  ; PLC PANEL SPARE 02
34    LD      M117  ; PLC PANEL SPARE 03
      OUT     Y41  ; PLC PANEL SPARE 03
36    LD      M118  ; PLC PANEL SPARE 04
      OUT     Y42  ; PLC PANEL SPARE 04
38    LD      M119  ; PLC PANEL SPARE 05
      OUT     Y43  ; PLC PANEL SPARE 05
40    LD      M120  ; MACH  UNIT-2 BND MANUAL CLMP CYL
      OUT     Y44  ; MACH UNIT-2 BNDG AUTO CLAMP CYL
42    LD      M121  ; MACH  UNIT-2 BND MANUAL CLMP CYL
      OUT     Y45  ; MACH  UNIT-2 BND MANUAL CLMP CYL
44    LD      M122  ; MACH  UNIT-3 BND MANUAL CLMP CYL
      OUT     Y46  ; MACH  UNIT-3 BND MANUAL CLMP CYL
46    LD      M123  ; MACH  UNIT-3 BND MANUAL CLMP CYL
      OUT     Y47  ; MACH  UNIT-3 BND MANUAL CLMP CYL
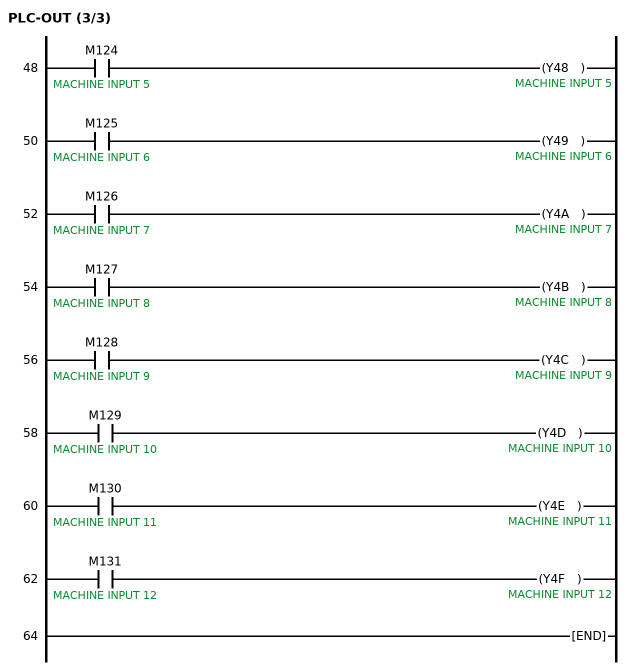
48    LD      M124  ; MACHINE INPUT 5
      OUT     Y48  ; MACHINE INPUT 5
50    LD      M125  ; MACHINE INPUT 6
      OUT     Y49  ; MACHINE INPUT 6
52    LD      M126  ; MACHINE INPUT 7
      OUT     Y4A  ; MACHINE INPUT 7
54    LD      M127  ; MACHINE INPUT 8
      OUT     Y4B  ; MACHINE INPUT 8
56    LD      M128  ; MACHINE INPUT 9
      OUT     Y4C  ; MACHINE INPUT 9
58    LD      M129  ; MACHINE INPUT 10
      OUT     Y4D  ; MACHINE INPUT 10
60    LD      M130  ; MACHINE INPUT 11
      OUT     Y4E  ; MACHINE INPUT 11
62    LD      M131  ; MACHINE INPUT 12
      OUT     Y4F  ; MACHINE INPUT 12
64    END
END_PROGRAM

PROGRAM ROBOT
